# EPICS IOC start-up script: acalcout/test.iocsh
dbLoadRecords("xaxis.db")
